// TwinCAT 3 PLC project Oefening2
// ProgramVersion: 3.1.4023.0
// libraries:
//   Tc2_BABasic, * (Beckhoff Automation GmbH)
//   Tc2_Standard, * (Beckhoff Automation GmbH)
//   Tc2_System, * (Beckhoff Automation GmbH)
//   Tc2_Utilities, * (Beckhoff Automation GmbH)
//   Tc3_Module, * (Beckhoff Automation GmbH)
// project tree:
//   / GlobalTextList.TcGTLO, PlcTask.TcTTO, Visualization Manager.TcVMO (not stored)
//   POUs/ FB_Knipperlicht.TcPOU, MAIN.TcPOU
//   VISUs/ Oefening2_VISU.TcVIS
// (motion and I/O tree: see PLC project oefening1)
// real-time tasks:
//   TASK PlcTask: cycle T#10ms, priority 20, ADS port 350
//   TASK PlcTask1: cycle T#10ms, priority 21, ADS port 351
//   TASK PlcTask2: cycle T#10ms, priority 22, ADS port 352
//   TASK PlcTask3: cycle T#10ms, priority 23, ADS port 353
//   TASK PlcTask4: cycle T#10ms, priority 24, ADS port 354
//   TASK PlcTask5: cycle T#10ms, priority 25, ADS port 355

CONFIGURATION Oefening2
    RESOURCE PLC ON TwinCAT3
        TASK PlcTask(INTERVAL := T#10ms, PRIORITY := 21);
        PROGRAM MAIN WITH PlcTask : MAIN;
    END_RESOURCE
END_CONFIGURATION

// ---- POUs/MAIN.TcPOU
PROGRAM MAIN

VAR_INPUT
	schakelaar_1 : BOOL;
	schakelaar_2 : BOOL;
	schakelaar_3 : BOOL;
END_VAR

VAR_OUTPUT
	kantoorlicht : BOOL;
END_VAR

VAR
	// CONTROLS THE INPUT
	START : INT;
	
	// Variable that checks the hour
	hourToStop : WORD;
	
	// F_TRIG
	F_TRIG : F_TRIG;
	
	// TwinCAT FB
	FB_LocalSystemTime : FB_LocalSystemTime;
	FB_ShortLongClick: FB_ShortLongClick;
	FB_SingleDoubleClick : FB_SingleDoubleClick;

	// Eigen FB
	Knipperlicht : FB_Knipperlicht;
END_VAR

FB_SingleDoubleClick(bSwitch:= schakelaar_1, tSwitchTime:= T#1S);

IF FB_SingleDoubleClick.bSingleClick THEN
	START := 1;
	Knipperlicht.CyclesReset := FALSE;
END_IF

IF (START > 0) THEN
	schakelaar_1 := FALSE;
	FB_LocalSystemTime(bEnable:= TRUE);
	kantoorlicht := TRUE;
	IF (FB_LocalSystemTime.systemTime.wMinute >= hourToStop) AND (Knipperlicht.Cycles <= 3) THEN
		Knipperlicht(Enable:= TRUE, OnTime:= T#500MS, OfTime:= T#500MS, Q=> kantoorlicht);
	ELSIF (Knipperlicht.Cycles > 3) THEN
		Knipperlicht(Enable:= TRUE, OnTime:= T#30S, OfTime:= T#0S, Q=> kantoorlicht);
		F_TRIG(CLK:= Knipperlicht.Q);
		
		IF FB_SingleDoubleClick.bDoubleClick THEN
			START := 2;
		END_IF
		
		IF (START > 1) THEN
			kantoorlicht := TRUE;
			FB_ShortLongClick(bSwitch:= schakelaar_1, tSwitchTime:= T#100MS);
			IF FB_ShortLongClick.bLongClick THEN
				START := 0;
			END_IF
		ELSIF F_TRIG.Q THEN
			START := 0;
		END_IF
	END_IF

ELSE
	schakelaar_1 := FALSE;
	kantoorlicht := FALSE;
	Knipperlicht(Enable:= TRUE, CyclesReset:=TRUE);
	
	IF schakelaar_3 THEN
		schakelaar_2 := FALSE;
		hourToStop := hourToStop + 1;
		schakelaar_3 := FALSE;
	ELSIF schakelaar_2 THEN
		schakelaar_3 := FALSE;
		hourToStop := hourToStop - 1;
		schakelaar_2 := FALSE;
	END_IF
END_IF;

END_PROGRAM

// ---- POUs/FB_Knipperlicht.TcPOU
FUNCTION_BLOCK FB_Knipperlicht
VAR_INPUT
	Enable : BOOL;	(* activatie knipperlicht*)
	OnTime : TIME;  (* tijd dat de lamp aan is *)
	OfTime : TIME;  (* tijd dat de lamp uit is *)
	CyclesReset : BOOL;
END_VAR

VAR_OUTPUT
	Q: BOOL;		(* het knipperlicht *)
	Freq: REAL;		(* de knipperfrequentie *)
	Duty: REAL;     (* de verhouding aan/totale-tijd *)
	Cycles: INT;	(* Hoeveelheid cycles voltooid *)
END_VAR

VAR
	Counter : BOOL;
	R_TRIG : R_TRIG;
	tOnTime: TOF;
	tOfTime: TON;
	tTotalTime: TIME; 
END_VAR

IF Enable THEN
	IF CyclesReset THEN
		Cycles := 0;
	ELSE
	tTotalTime := OnTime + OfTime;
	Duty := (TIME_TO_REAL(OnTime)/(TIME_TO_REAL(OnTime)+TIME_TO_REAL(OfTime))*100);
	Freq := 1000 / (TIME_TO_REAL(OnTime)+TIME_TO_REAL(OfTime));
	
	tOnTime(IN:= NOT tOfTime.Q  , PT:= OnTime, Q=>Q);
	tOfTime(IN:= tOntime.Q 	    , PT:= OfTime, Q=>Q);
	
	R_TRIG(CLK:= Q, Q=> Counter);
	Cycles := Cycles + BOOL_TO_INT(Counter);
	END_IF
ELSE
	Q := FALSE;
END_IF

END_FUNCTION_BLOCK

// ---- VISUs/Oefening2_VISU.TcVIS
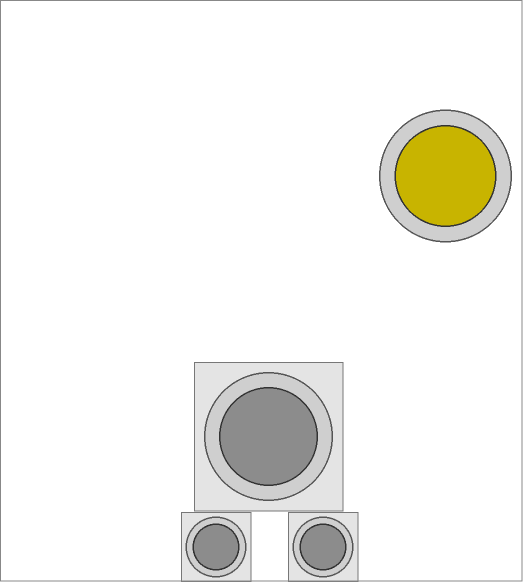
VISUALIZATION Oefening2_VISU  // 523x582
    Lamp1 (368,99 155x154), variable: MAIN.kantoorlicht, style: Lamp-Lamp1-Yellow
    PushSwitch (194,359 149x155), variable: MAIN.schakelaar_1, behaviour: TOGGLE, style: Switch-PushSwitch-Gray
    PushSwitch (181,512 70x70), variable: MAIN.schakelaar_2, behaviour: TOGGLE, style: Switch-PushSwitch-Gray
    PushSwitch (288,512 70x70), variable: MAIN.schakelaar_3, behaviour: TOGGLE, style: Switch-PushSwitch-Gray
END_VISUALIZATION
